FUNCTION_BLOCK Axis IMPLEMENTS I_AXIS
VAR_IN_OUT CONSTANT
	cMinPos : LREAL;
	cMaxPos: LREAL;
END_VAR
VAR_INPUT
	bEnable : BOOL;
	bHalt : BOOL;
	bStop : BOOL;
	bReset : BOOL;
END_VAR
VAR_OUTPUT
	axisRef : AXIS_REF;
	fbMcReadStatus : MC_ReadStatus;
END_VAR
VAR
	bCalibrationCam AT%I* :  BOOL;
	
	//Data for coupling operations
	//--------------------------------------------------------------
	
	slaveAxis : REFERENCE TO AXIS_REF;
	slaveStatus : REFERENCE TO ST_AXISSTATUS;
	lrRatioNumerator : LREAL := 1;
	uiRatioDenominator : UINT := 1;
	
	//--------------------------------------------------------------
	
	fbMcHome : MC_Home;
	fbMcGearIn : MC_GearIn;
	fbMcGearOut : MC_GearOut;
	
	fbMcPower : MC_Power;
	fbMcHalt : MC_Halt;
	fbMcStop : MC_Stop;
	fbMcReset : MC_Reset;
	fbMcMoveAbsolute : MC_MoveAbsolute;
	
END_VAR

fbMcMoveAbsolute(
	Axis:= axisRef, 
	Velocity:= 200, 
);


fbMcStop(
	Axis:= axisRef, 
	Execute:= bStop
);
	
fbMcHalt(
	Axis:= axisRef, 
	Execute:= bHalt
);
	
fbMcReset(
	Axis:= axisRef, 
	Execute:= bReset
);
	
fbMcPower(
	Axis:= axisRef, 
	Enable:= bEnable, 
	Enable_Positive:= bEnable, 
	Enable_Negative:= bEnable, 
	Override:= , 
	BufferMode:= , 
	Options:= , 
	Status=> , 
	Busy=> , 
	Active=> , 
	Error=> , 
	ErrorID=> 
);

fbMcReadStatus(
	Axis:= axisRef, 
	Enable:= TRUE, 
);

fbMcHome(
	Axis:= axisRef, 
	bCalibrationCam:= bCalibrationCam, 
);

IF 		__ISVALIDREF(slaveAxis)
	AND __ISVALIDREF(slaveStatus)
THEN

	fbMcGearIn(
		Master:= axisRef, 
		Slave:= slaveAxis, 
		RatioNumerator:= lrRatioNumerator, 
		RatioDenominator:= uiRatioDenominator
	);
	
	IF NOT fbMcGearIn.Busy
	THEN
		fbMcGearIn.Execute := FALSE;
	END_IF
	
	
	fbMcGearOut(Slave:= slaveAxis);
	IF NOT fbMcGearOut.Busy
	THEN
		fbMcGearOut.Execute := FALSE;
	END_IF
	
END_IF


IF fbMcHome.Done
THEN
	fbMcHome.Execute := FALSE;
END_IF

METHOD MoveAbsolute
VAR_INPUT
	lrPosition : LREAL;
END_VAR
IF lrPosition < cMinPos OR lrPosition > cMaxPos
THEN
	RETURN;
END_IF
fbMcMoveAbsolute(Axis := axisRef, Execute := TRUE , Position := lrPosition);
fbMcMoveAbsolute.Execute := FALSE;
END_METHOD

METHOD PrepareCoupling : I_Axis
VAR_INPUT
	slaveAxis : REFERENCE TO AXIS_REF;
	slaveStatus : REFERENCE TO ST_AXISSTATUS;
	lrRatioNumerator : LREAL;
	uiRatioDenominator : UINT;
END_VAR
PrepareCoupling := THIS^;
THIS^.slaveAxis REF= slaveAxis;
THIS^.slaveStatus REF= slaveStatus;
THIS^.lrRatioNumerator := lrRatioNumerator;
THIS^.uiRatioDenominator := uiRatioDenominator;
END_METHOD

METHOD PrepareDecoupling : I_Axis
VAR_INPUT
	slaveAxis : REFERENCE TO AXIS_REF;
	slaveStatus : REFERENCE TO ST_AXISSTATUS;
END_VAR
PrepareDecoupling := THIS^;
THIS^.slaveAxis REF= slaveAxis;
THIS^.slaveStatus REF= slaveStatus;
END_METHOD

METHOD StartCoupling : I_Axis
VAR_INPUT
END_VAR
StartCoupling := THIS^;
IF NOT __ISVALIDREF(slaveStatus)
THEN
	RETURN;
END_IF

IF NOT slaveStatus.Coupled
THEN
	fbMcGearIn.Execute := TRUE;
END_IF
END_METHOD

METHOD StartDecoupling : BOOL
VAR_INPUT
END_VAR

IF NOT __ISVALIDREF(slaveStatus)
THEN
	RETURN;
END_IF

IF slaveStatus.Coupled
THEN
	fbMcGearOut.Execute := TRUE;
ELSE
	StartDecoupling := TRUE;
END_IF
END_METHOD

METHOD StartHoming : BOOL;
VAR_INPUT
END_VAR
IF NOT fbMcGearIn.Execute
	//AND fbMcReadStatus.Valid
	//AND NOT fbMcReadStatus.Status.Homed 
THEN
	
	fbMcHome.Execute := TRUE;
	IF fbMcHome.Busy
	THEN
		fbMcHome.Execute := FALSE;
		StartHoming := TRUE;
	END_IF
	
END_IF
END_METHOD

END_FUNCTION_BLOCK

(* stored: Version 1.1.0.1, ProductVersion 3.1.4024.2
   POU Axis: Id {24fff4e6-e39f-4350-bd18-ef00f5f91f03}, SpecialFunc None
   Method MoveAbsolute: Id {f47e21c3-cef3-4c6f-a3be-54a65a02bcdb}
   Method PrepareCoupling: Id {d7878975-8fc9-40ec-8586-907322a90143}
   Method PrepareDecoupling: Id {21d52ac6-f4dc-441d-aadf-f3c53372b8fe}
   Method StartCoupling: Id {33e91c27-060b-4aba-a2bf-d064c83cf754}
   Method StartDecoupling: Id {4837a0df-aaef-47d5-97eb-083f968790d7}
   Method StartHoming: Id {d6df9a82-84a4-4ac0-b48c-1d732d0b93bd} *)
